TYPE ST_Config :
STRUCT
  bEnabled : BOOL;
  nValue : INT;
END_STRUCT
END_TYPE

(* stored: Version 1.1.0.1, ProductVersion 3.1.4024.12
   DUT ST_Config: Id {aaaaaaaa-bbbb-cccc-dddd-eeeeeeeeeeee} *)
